FUNCTION F_ArrayStr : ARRAY [1..NO_OF_STRING_PARAM] OF STRING
VAR_INPUT
	sParam		: ARRAY [1..NO_OF_STRING_PARAM] OF STRING;
	sParam1		: STRING;
	//sParam		: ARRAY [1..NO_OF_STRING_PARAM] OF STRING;
	//bParam		: ARRAY [1..NO_OF_BOOL_PARAM] OF BOOL;
	//dParam		: ARRAY [1..NO_OF_LREAL_PARAM] OF LREAL;
END_VAR

	F_ArrayStr := sParam;
	F_ArrayStr[1] := sParam1;

END_FUNCTION

(* stored: Version 1.1.0.1, ProductVersion 3.1.4022.18
   POU F_ArrayStr: Id {e6a20e00-302a-4e85-bce9-2258f07541d2}, SpecialFunc None *)
